FUNCTION_BLOCK ClockTicker (* Basic Function Block Type *)
  (* Standard: 61499-2 *)
  (* Version 0.2, 2003-12-04, JHC, Rockwell Automation, Renamed for better indexing. *)
  (* Compiler header: package fb.rt.wago; #include <sys/time.h> *)
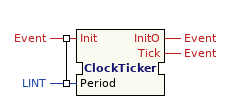
  EVENT_INPUT
    Init WITH Period; (* Initialization Request *)
  END_EVENT
  EVENT_OUTPUT
    InitO; (* Initialization Confirm *)
    Tick; (* Execution Confirmation *)
  END_EVENT
  VAR_INPUT
    Period : LINT; (* Period in us *)
  END_VAR
  VAR
    ClockTimedOut : BOOL;
    theclock : DATE_AND_TIME;
  END_VAR
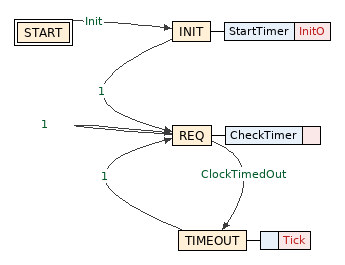
  EC_STATES
    START; (* Initial State *)
    INIT : StartTimer -> InitO; (* Initialization *)
    REQ : CheckTimer; (* Normal execution *)
    TIMEOUT : -> Tick;
  END_STATES
  EC_TRANSITIONS
    START TO INIT := Init;
    INIT TO REQ := 1;
    REQ TO TIMEOUT := ClockTimedOut;
    TIMEOUT TO REQ := 1;
    REQ TO REQ := 1;
  END_TRANSITIONS
  ALGORITHM StartTimer IN C: (* Initialization algorithm *)
gettimeofday(&me->theclock, NULL);
  END_ALGORITHM
  ALGORITHM CheckTimer IN C: (* Normally executed algorithm *)
struct timeval timenow, timediff;
long long result;

gettimeofday(&timenow, NULL);
timersub(&timenow, &me->theclock, &timediff);
result = (long long)(timediff.tv_sec) * 1000000 + timediff.tv_usec;

if( result > me->Period )
{
 me->ClockTimedOut = true;
 gettimeofday(&me->theclock, NULL);
}
  END_ALGORITHM
END_FUNCTION_BLOCK
